Staubli VAL3: tool.pjx

--- tool.pjx ---
Parameters version=s7.6.1 stackSize=5000 millimeterUnit=true
Program file=buildList.pgx
Program file=editAction.pgx
Program file=editTool.pgx
Program file=insertInstr.pgx
Program file=listAdd.pgx
Program file=loadPage.pgx
Program file=main.pgx
Program file=onBackSpace.pgx
Program file=onEnterEvent.pgx
Program file=onExit.pgx
Program file=onF1Event.pgx
Program file=onF2Event.pgx
Program file=onF3Event.pgx
Program file=onF4Event.pgx
Program file=onF5Event.pgx
Program file=onF6Event.pgx
Program file=onF7Event.pgx
Program file=onF8Event.pgx
Program file=onStart.pgx
Program file=refresh.pgx
Program file=refreshAction.pgx
Program file=refreshDynamic.pgx
Program file=refreshStatic.pgx
Data file=tool.dtx
Library alias=events path=Disk://..//templates/instruction/instruction.pjx
Library alias=page path=Disk://kernel/template/page/page.pjx
Library alias=use path=Disk://kernel/userPage/userPage.pjx
Library alias=language path=Disk://kernel/language/language.pjx
Library alias=saveData path=Disk://saveData/saveData.pjx
Library alias=tcp path=Disk://kernel/tool/tool.pjx
Library alias=cycleStatus path=Disk://cycleStatus/cycleStatus.pjx
Type name=InstrItem path=Disk://kernel/template/InstrItem/InstrItem.pjx
Type name=FrameItem path=Disk://kernel/template/FrameItem/FrameItem.pjx

--- tool.dtx ---
num nIndex
num nIndexTool
num nKey
public num nPage
num nRefresh
num nTime = 1
num nView
string sEvent
public string sItems
string sList
string sMenu
string sMessage
string sMenu8[8]
string sActionON[3]
string sActionOFF[3]
bool bButton[8]
bool bLarge
InstrItem iInstrTcpON[3]
  [0]
    string sType
    string sData
  [1]
    string sType
    string sData
  [2]
    string sType
    string sData
InstrItem iInstrTcpOFF[3]
  [0]
    string sType
    string sData
  [1]
    string sType
    string sData
  [2]
    string sType
    string sData
tool tTool = {fatherId=flange[0], ioLink=valve1}
string sSession
frame fFrame = {fatherId=world[0]}

--- main.pgx ---
public program main()
  local num l_nSize
  local bool l_bSave
  local num l_nStatus
  local bool l_bToReset
  local bool l_bCalcolate
  local frame l_fNewWorld
begin
  // INIT
  call onStart()
  // LOOP UNTIL nKey=255
  do
    call tcp:getSize(l_nSize)
    call tcp:getTool(tTool,nIndexTool)
    call refresh()
    if l_bCalcolate
      fFrame.trsf=saveData:fFrameItem[saveData:nFrameActive].fFrame.trsf
      $jogContext(tTool,fFrame,0)
      l_bCalcolate=false
    endIf
    nKey=get()
    // tool setting
    if !cycleStatus:bCycle
      if !(cycleStatus:nWorkingMode==1 and (cycleStatus:nWorkingStatus==6 or cycleStatus:nWorkingStatus==0))
        l_bToReset=true
      else
        if l_bToReset
          resetMotion()
          l_bToReset=false
        endIf
      endIf
    endIf
    // list....
    call use:listevent(nKey,nIndex,sEvent)
    nView=use:nView
    switch nKey
      case 263
        // BACKSPACE
        call onBackSpace(tTool)
        l_bCalcolate=true
        l_bSave=true
      break
      case 264
        // LEFT CLICK -1
        if nIndexTool>0
          nIndexTool=nIndexTool-1
          l_bSave=true
          l_bCalcolate=true
        endIf
      break
      case 268
        // RIGHT CLICK +1
        if nIndexTool<l_nSize-1
          nIndexTool=nIndexTool+1
          l_bSave=true
          l_bCalcolate=true
        endIf
      break
      case 271
        call onF1Event()
      break
      case 272
        call onF2Event()
      break
      case 273
        // HERE
        call onF3Event(l_bSave)
      break
      case 274
        // COMPUTE
        call onF4Event(l_bSave)
        l_bCalcolate=true
      break
      case 275
        // MOVE
        call onF5Event()
      break
      case 276
        // DUPLICATE
        call onF6Event(tTool,l_bSave)
      break
      case 277
        // DELETE
        call onF7Event(l_bSave)
      break
      case 278
        // NEW
        call onF8Event(l_bSave)
      break
      case 270
        // USE ALSO BACKSPACE
        // EDIT FIELD
        call onEnterEvent(tTool)
        l_bCalcolate=true
        l_bSave=true
      break
    endSwitch
  until nKey==255
  // on Exit
  fFrame.trsf=saveData:fFrameItem[saveData:nFrameActive].fFrame.trsf
  $jogContext(tTool,fFrame,0)
  call onExit(l_bSave)
end

--- buildList.pgx ---
program buildList()
  local num l_nSize
  local string l_sName
  local num i
  local string l_sMessage
  local tool l_tTool
  local string l_sEmpty
  local string l_sItem
begin
  // INIT the list
  l_sEmpty=""
  call use:stringCopy(l_sEmpty,sList)
  //
  // Build the list
  //
  // get the GUN
  call tcp:getTool(l_tTool,nIndexTool)
  // show the gun
  call tcp:getName(l_sName,nIndexTool)
  call language:message(l_sMessage,21)
  l_sName=l_sMessage+"> "+l_sName
  // create the list
  call listAdd(l_sName)
  l_sItem=("coord  X > "+toString(".2",l_tTool.trsf.x))
  call listAdd(l_sItem)
  l_sItem=("coord  Y > "+toString(".2",l_tTool.trsf.y))
  call listAdd(l_sItem)
  l_sItem=("coord  Z > "+toString(".2",l_tTool.trsf.z))
  call listAdd(l_sItem)
  l_sItem=("coord RX > "+toString(".2",l_tTool.trsf.rx))
  call listAdd(l_sItem)
  l_sItem=("coord RY > "+toString(".2",l_tTool.trsf.ry))
  call listAdd(l_sItem)
  l_sItem=("coord RZ > "+toString(".2",l_tTool.trsf.rz))
  call listAdd(l_sItem)
  // TCP ON OFF
  call language:message(l_sMessage,123)
  call use:strfill(l_sMessage,9,l_sMessage)
  l_sItem=l_sMessage+">ON  "+toString("",l_tTool.otime)+ "mm"
  call listAdd(l_sItem)
  l_sItem=l_sMessage+">OFF "+toString("",l_tTool.ctime)+ "mm"
  call listAdd(l_sItem)
end

--- editAction.pgx ---
program editAction(InstrItem& x_iAction[], bool& x_bSave[], num& x_nTime)
  local string l_sMessage
  local string l_sInstruction
  local bool l_bYes
  local num i
  local num l_nKey
  local num l_nIndex
  local string l_sButton[2]
  local string l_sEmpty
  local num l_nTime
  local InstrItem l_iAction[3]
  local InstrItem l_iNewAction
  local string l_sEvent
begin
  // make a copy
  l_nTime=x_nTime
  for i=0 to size(x_iAction)-1
    // copy all the action
    l_iAction[i]=x_iAction[i]
  endFor
  // loop
  do
    // refresh
    call refreshAction(l_nIndex,l_iAction,l_nTime)
    // get the Key
    l_nKey=get()
    l_sEmpty=""
    call use:listevent(l_nKey,l_nIndex,l_sEvent)
    if l_nKey==270
      switch l_nIndex
        case 0,1,2
          //
          //  edit the instruction
          //
          // insert a new one
          if l_iAction[l_nIndex].sType==""
            l_iNewAction.sType=l_iAction[l_nIndex].sType
            call insertInstr(l_iNewAction)
            if l_iNewAction.sData!=""
              l_iAction[l_nIndex]=l_iNewAction
            endIf
          else
            // delete
            call language:message(l_sMessage,171)
            // get the yes_no button
            call language:getYesNo(l_sButton)
            // ask the question
            call use:yes_no(l_sMessage,l_sButton,l_bYes)
            if l_bYes
              l_iAction[l_nIndex].sType=""
              l_iAction[l_nIndex].sData=""
            endIf
          endIf
        break
        case 3
          //
          // set the distance...
          //
          call use:findPos(l_sEvent,">",i)
          // clean the line
          call use:listcursor(use:nView,false)
          // edit it
          l_sEmpty=""
          call use:changeValue(l_nTime,-300,300,i+use:nTopX+3,use:nView+use:nTopY+1,l_sEmpty)
        break
      endSwitch
    endIf
    // use left to go bak or escape to no validate
  until l_nKey==264 or l_nKey==255 or l_nKey==278
  //
  if l_nKey!=255
    x_bSave=true
    for i=0 to size(x_iAction)-1
      // copy all the action
      x_iAction[i]=l_iAction[i]
    endFor
    x_nTime=l_nTime
  endIf
  //nullKey
  call use:nullKey(nKey)
end

--- editTool.pgx ---
program editTool(tool& x_tTool)
  local num i
  local num l_nX
  local num l_nY
  local bool l_bEdit
  local string l_sEmpty
  local tool l_tTool
  local num l_nTime
begin
  //
  //  search the ">" to change the right side from here of the the string
  //
  call use:getListPosition(l_nX,l_nY)
  //i=find(sEvent,">")
  call use:findPos(sEvent,">",i)
  // clean the line
  call use:listcursor(use:nView,false)
  // read the name
  if i!=-1 and nIndex==0
    sEvent=right(sEvent,getDisplayLen(sEvent)-i-2)
    // read the name
    call use:read(i+l_nX+1,1,sEvent,10,false)
  endIf
  // COPY
  l_sEmpty=""
  l_tTool=x_tTool
  l_tTool.otime=x_tTool.otime
  l_tTool.ctime=x_tTool.ctime
  // INDEX
  switch nIndex
    case 0
      if nIndexTool!=-1
        call tcp:setName(sEvent,nIndexTool)
      endIf
    break
    case 1
      //
      //  x-value
      //
      call use:changeValue(l_tTool.trsf.x,0,0,i+40-use:nBottomX+1,use:nView+1,l_sEmpty)
    break
    case 2
      //
      //  y-value
      //
      call use:changeValue(l_tTool.trsf.y,0,0,i+40-use:nBottomX+1,use:nView+1,l_sEmpty)
    break
    case 3
      //
      //  z-value
      //
      call use:changeValue(l_tTool.trsf.z,0,0,i+40-use:nBottomX+1,use:nView+1,l_sEmpty)
    break
    case 4
      //
      //  rx-value
      //
      call use:changeValue(l_tTool.trsf.rx,0,0,i+40-use:nBottomX+1,use:nView+1,l_sEmpty)
    break
    case 5
      //
      //  ry-value
      //
      call use:changeValue(l_tTool.trsf.ry,0,0,i+40-use:nBottomX+1,use:nView+1,l_sEmpty)
    break
    case 6
      //
      //  rz-value
      //
      call use:changeValue(l_tTool.trsf.rz,0,0,i+40-use:nBottomX+1,use:nView+1,l_sEmpty)
    break
    case 7
      //
      // change the ACTION ON
      //
      l_nTime=l_tTool.otime
      call editAction(iInstrTcpON,l_bEdit,l_nTime)
      if l_bEdit
        call tcp:setInstr(iInstrTcpON,nIndexTool,true)
        l_tTool.otime=l_nTime
      endIf
    break
    case 8
      //
      // change the ACTION OFF
      //
      l_nTime=l_tTool.ctime
      call editAction(iInstrTcpOFF,l_bEdit,l_nTime)
      if l_bEdit
        call tcp:setInstr(iInstrTcpOFF,nIndexTool,false)
        l_tTool.ctime=l_nTime
      endIf
    break
  endSwitch
  // copy back
  x_tTool.trsf=l_tTool.trsf
  x_tTool.otime=l_tTool.otime
  x_tTool.ctime=l_tTool.ctime
end

--- insertInstr.pgx ---
program insertInstr(InstrItem& x_iItem[])
  local num i
  local num l_nIndex
  local string l_sPath
  local string l_sItem
begin
  // TODO
  call use:setSizeList(14,0,10,11)
  call use:setView(false)
  call use:listcreate("Select")
  // insert the action on Point
  call use:listadd(saveData:sInstrOnPoint)
  call use:listupdate(0)
  // SELECT THE ITEM
  do
    i=get()
    call use:listevent(i,l_nIndex,l_sItem)
  until i==255 or i==270
  // copy
  x_iItem.sType=l_sItem
  // define it
  if x_iItem.sType!="" and i==270
    // load the instruction
    call saveData:getPathInstr(x_iItem.sType,l_sPath)
    // load the instruction
    events:libLoad(l_sPath)
    delay(0)
    call events:onInsert(x_iItem.sData)
    // insert the item
    return
  endIf
  // NOT GOOD
  x_iItem.sType=""
  x_iItem.sData=""
end

--- onBackSpace.pgx ---
program onBackSpace(tool& x_tTool[])
begin
  //
  // NB sEvent is the selected
  // element in the LIST
  //
  if nIndex==0
    call editTool(x_tTool)
    call tcp:setTool(x_tTool,nIndexTool)
    logMsg("[KERNEL] INTERFACE:Change value of the tool :"+toString("",nIndexTool))
  endIf
  //
end

--- onEnterEvent.pgx ---
program onEnterEvent(tool& x_tTool[])
begin
  //
  // NB sEvent is the selected
  // element in the LIST
  //
  call editTool(x_tTool)
  call tcp:setTool(x_tTool,nIndexTool)
  logMsg("[KERNEL] INTERFACE:Change value of the tool :"+toString("",nIndexTool))
  //
end

--- onExit.pgx ---
program onExit(bool x_bSave)
  local string l_sMessage
  local bool l_bYes
  local num l_nResult
begin
  if x_bSave
    // ask to save
    //    call language:message(l_sMessage,-1)
    //    call use:yes_no(l_sMessage,l_bYes)
    //    if l_bYes
    call tcp:save(l_nResult)
    // send back the gun
    //    endIf
  endIf
  // give back and update
  saveData:nIndexTool=nIndexTool
  call tcp:getTool(saveData:tTool,nIndexTool)
end

--- onF3Event.pgx ---
program onF3Event(bool x_bSave)
  local string l_sMessage
  local bool l_bYes
  local string l_sButton[2]
begin
  // look if the bButton is enable
  if bButton[2]
    //
    if !cycleStatus:bCycle and nIndexTool==0
      call language:message(l_sMessage,125)
      // get the yes_no button
      call language:getYesNo(l_sButton)
      // ask the question
      call use:yes_no(l_sMessage,l_sButton,l_bYes)
      if l_bYes
        call tcp:here()
        call language:message(l_sMessage,121)
        popUpMsg(l_sMessage)
        logMsg("[KERNEL] INTERFACE:Take the reference point")
        x_bSave=true
      endIf
    endIf
  endIf
end

--- onF4Event.pgx ---
program onF4Event(bool& x_bSave[])
  local bool l_bCheck
  local string l_sMessage
  local frame l_fNewWorld
begin
  // look if the bButton is enable
  if bButton[3]
    //
    if !cycleStatus:bCycle
      if nIndexTool!=0
        call tcp:checkPoint(l_bCheck)
        if l_bCheck
          call tcp:compose(nIndexTool)
          call tcp:getTool(tTool,nIndexTool)
          fFrame=saveData:fFrameItem[saveData:nFrameActive].fFrame
          $jogContext(tTool,fFrame,0)
          logMsg("[KERNEL] INTERFACE:Compose the TCP")
          x_bSave=true
        else
          call language:message(l_sMessage,122)
          popUpMsg(l_sMessage)
        endIf
      endIf
    endIf
  endIf
end

--- onF5Event.pgx ---
program onF5Event()
  local bool l_bCheck
  local string l_sMessage
begin
  // look if the bButton is enable
  if bButton[4]
    //
    if !cycleStatus:bCycle and workingMode()==1
      resetMotion()
      call tcp:checkPoint(l_bCheck)
      if l_bCheck
        call language:message(l_sMessage,203)
        call tcp:goToPoint(nIndexTool)
        logMsg("[KERNEL] INTERFACE:Go to the reference Point")
        call use:timerDialog(l_sMessage,2)
      endIf
    endIf
  endIf
end

--- onF6Event.pgx ---
program onF6Event(tool x_tTool, bool& x_bSave[])
  local string l_sMessage
  local string l_sName
  local num l_nSize
begin
  // look if the bButton is enable
  if bButton[5]
    //
    // DUPLICATE
    //
    call language:message(l_sMessage,126)
    call tcp:getName(l_sName,nIndexTool)
    popUpMsg(l_sMessage+l_sName)
    call tcp:new(x_tTool.trsf)
    call tcp:getSize(l_nSize)
    nIndexTool=l_nSize-1
    //    // refresh and modify the name
    call buildList()
    call refreshStatic()
    nIndex=0
    call editTool(x_tTool)
    logMsg("[KERNEL] INTERFACE:Insert new tool at index: "+toString("",l_nSize))
    x_bSave=true
  endIf
end

--- onF7Event.pgx ---
program onF7Event(bool& x_bSave[])
  local string l_sMessage
  local bool l_bFound
  local string l_sTrajName
  local bool l_bYes
  local string l_sString
  local string l_sButton[2]
begin
  // look if the bButton is enable
  if bButton[6]
    // delete the selected tool

  endIf
end

--- onF8Event.pgx ---
program onF8Event(bool& x_bSave[])
  local num l_nSize
  local tool l_tEmpty
begin
  // look if the bButton is enable
  if bButton[7]
    //
    l_tEmpty=flange
    call tcp:new(l_tEmpty.trsf)
    call tcp:getSize(l_nSize)
    nIndexTool=l_nSize-1
    // refresh and modify the name
    call buildList()
    call refreshStatic()
    nIndex=0
    sEvent=""
    call editTool(l_tEmpty)
    logMsg("[KERNEL] INTERFACE:Insert new tool at index: "+toString("",l_nSize))
    x_bSave=true
  endIf
end

--- onStart.pgx ---
program onStart()
  local num i
  local string l_sMessage
begin
  // logMsg
  logMsg("[KERNEL] INTERFACE:PAGE TOOL")
  // be aware these value will change all the value
  call language:message(l_sMessage,129)
  popUpMsg(l_sMessage)
  // set the tool as default
  nIndexTool=saveData:nIndexTool
  // reset the Key pressure
  call use:nullKey(nKey)
  // define the list
  call buildList()
  // build the page
  call refreshStatic()
  // define the list
end

--- refresh.pgx ---
program refresh()
// // page refresh
begin
  // refresh the static message
  if (nKey>=270 and nKey<=278) or nKey==268 or nKey==264 or use:bUseRefresh
    call buildList()
    call refreshStatic()
    call refreshDynamic()
  else
    // refresh the Dynamic message
    if abs(clock()-nRefresh)>nTime
      call refreshDynamic()
    endIf
  endIf
end

--- refreshAction.pgx ---
program refreshAction(num x_nIndex, InstrItem& x_iAction[], num x_nDistance)
  local string l_sMessage
  local string l_sTitle
  local num i
  local string l_sAction
  local num l_nSize
begin
  //
  // INSTRUCTION
  //
  cls()
  // create a menu to edit the action
  call use:setSizeList(5,3,30,4)
  call use:setView(false)
  // show the title
  call tcp:getSize(l_nSize)
  call language:message(l_sMessage,124)
  l_sTitle=l_sMessage+toString("3",nIndexTool)+"/"+toString("",l_nSize-1)
  call tcp:getName(l_sMessage,nIndexTool)
  l_sTitle=l_sTitle+" "+l_sMessage
  call use:listcreate(l_sTitle)
  // get the action string
  call language:message(l_sMessage,176)
  // insert all the 3 action
  for i=0 to 2
    l_sAction=l_sMessage+toString("",i+1)+"> "+x_iAction[i].sType+" "+x_iAction[i].sData
    call use:listadd(l_sAction)
  endFor
  call language:message(l_sMessage,177)
  l_sMessage=l_sMessage+"> "+toString("",x_nDistance)+" mm"
  call use:listadd(l_sMessage)
  // show it
  call use:clear(0,13)
  call use:typeMenu(8,"OK")
  use:nView=x_nIndex
  call use:listupdate(0)
  //
end

--- refreshStatic.pgx ---
program refreshStatic()
  local num l_nSize
  local string l_sMessage
  local string l_sTitle
  local string l_sInstruction
  local num i
begin
  cls()
  //
  // set the view of the use:nPage..
  //
  // SET THE use:nPage NUMBER
  use:nPage=1400
  //
  if nIndexTool==0
    use:nPage=use:nPage+6
  endIf
  if cycleStatus:bCycle
    use:nPage=use:nPage+3
  endIf
  // get the size
  call tcp:getSize(l_nSize)
  // USE <>PROFILE for <>nPage
  use:nPage=use:nPage+abs(limit(saveData:mode,0,2)-2)
  // load the menu page
  if saveData:language!="japanese"
    // SET THE VIEW OF THE PAGE
    call language:page(l_sMessage,use:nPage)
    // define the menu
    call use:stringToArray(l_sMessage,sMenu)
    // hide the new button
    if nIndexTool!=l_nSize-1 and size(sMenu)>1
      sMenu[7]=""
    endIf
    call use:setMenu(sMenu,true,2)
  else
    // japanese use the array for the menu
    call language:page(sMenu8,use:nPage)
    call use:stringCopy(sMenu8,sMenu)
    // hide the new button
    if nIndexTool!=l_nSize-1 and size(sMenu)>1
      sMenu[7]=""
    endIf
    call use:setMenu(sMenu,false,2)
  endIf
  //
  call use:getMenu(sMenu,bButton)
  //
  // CREATE THE LIST
  //
  // define your list size for default
  call use:setSizeList(19,0,19,9)
  call use:setView(bLarge)
  //
  call language:message(l_sTitle,124)
  l_sTitle=l_sTitle+toString("3",nIndexTool)+"/"+toString("",l_nSize-1)
  call use:listcreate(l_sTitle)
  // insert inside the list
  call use:listadd(sList)
  // show the instruction ON
  call tcp:getInstr(iInstrTcpON,true,nIndexTool)
  l_sInstruction=iInstrTcpON.sType+" "+iInstrTcpON.sData
  for i=1 to size(iInstrTcpON)-1
    l_sInstruction=l_sInstruction+"·"+iInstrTcpON[i].sType+" "+iInstrTcpON[i].sData
  endFor
  call use:typeLen(0,11,"ON >"+l_sInstruction,40)
  // show the instruction OFF
  call tcp:getInstr(iInstrTcpOFF,false,nIndexTool)
  // array to string
  l_sInstruction=iInstrTcpOFF.sType+" "+iInstrTcpOFF.sData
  for i=1 to size(iInstrTcpOFF)-1
    l_sInstruction=l_sInstruction+"·"+iInstrTcpOFF[i].sType+" "+iInstrTcpOFF[i].sData
  endFor
  call use:typeLen(0,12,"OFF>"+l_sInstruction,40)
  //
  // refresh the cursor
  use:nView=nView
  // refresh the list
  call use:listupdate(nIndex-nView)
end
